FUNCTION_BLOCK FB_ElementA IMPLEMENTS I_VisitibleElement
VAR_INPUT
END_VAR
VAR_OUTPUT
END_VAR
VAR
END_VAR

METHOD accept
VAR_INPUT
	in_ipVisitor	: I_Visitor;
END_VAR
in_ipVisitor.VisitElementA(in_fbElementA:= THIS^);
END_METHOD

END_FUNCTION_BLOCK

(* stored: Version 1.1.0.1
   POU FB_ElementA: Id {9aa9f134-b544-4239-b9c4-046d9cb7361a}, SpecialFunc None
   Method accept: Id {6aa86e29-2a64-432c-94e6-33984946ac8b} *)
